FUNCTION_BLOCK Q_SelectColourMap (* Command Select Colour Map ( VT version 4 and later ) ( Part 6 - F.60 ) *)
  (* Standard: ISO 11783-6; Description: Copyright (c) 2022 HR Agrartechnik GmbH This program and the accompanying materials are made available under the terms of the Eclipse Public License 2.0 which is available at https://www.eclipse.org/legal/epl-2.0/ SPDX-License-Identifier: EPL-2.0 see Description Tab *)
  (* Version 1.0, 2022-07-08, Franz Höpfinger, HR Agrartechnik GmbH *)
  PACKAGE isobus::UT::Q;
  IMPORT isobus::UT::Q::const::IDs::ID_NULL;
  (* Documentation:
  Command Select Colour Map ( VT version 4 and later ) ( Part 6 - F.60 )
   The Select Colour Map command is used to select the active Colour Map. This command can take a long time to execute. The command applies to any presentation from the originating Working Set, which includes objects that may be shown on other Working Set screens (e.g. Auxiliary Control objects as may be presented on VT proprietary and other Working Set masks using the Auxiliary Control Designator Type 2 Object Pointer).
   Valid values for u16ObjIdColourMap
   The Select Colour Map or Palette command (F.60) carries, in bytes 2,3, the Object ID of the Colour Map object, the Colour Palette object, or FFFF16 to restore the default colour mapping (see A.3):
    - ColourMap: 39000 – 39999 (VT version 4 and later)
   - ColourPalette: 45000 – 45999 (VT version 6 and later, per Annex F.60)
   - FFFF16: restores the default colour table (see A.3)
    Implementation note (VTClientHelper): iso_is_colour_map_id only accepts the ColourMap range — a ColourPalette ID (45000 – 45999) is rejected. In addition, ID_NULL (65535), the documented FFFF16 value to restore the default colour table, is swallowed by cmd_select_colour_map_or_palette, which returns VT_E_NO_ERR (0) without sending any command to the VT. These are known deviations.
   param[in] {objectID, uint16_t}
   Object ID of Colour map object or FFFF to restore the default colour table (see A.3)
   Return Values (s16result):
   int16_t
    - VT_E_NO_ERR (0) - OK
   - VT_E_NOT_READY (-131) - VT client not yet ready
   - VT_E_OVERFLOW (-6) - buffer overflow
   - VT_E_NOACT (-8) - Command not possible in current state
   - VT_E_NO_INSTANCE (-21) - No VT client available
   - VT_E_ISO_INSTANCE_INVALID (-129) - Identifier for instance (connection) invalid
   - VT_E_NOT_ALIVE (-130) - Identifier for instance valid, but VT Dead.
   - VT_OK_BUFFERED (18) - command buffered, waiting for VT to be ready
    Instanz-Eindeutigkeit (Instance Uniqueness)
   Dieser Baustein ist konzeptionell als Singleton (genau eine Instanz im gesamten Programm) vorgesehen.
  *)
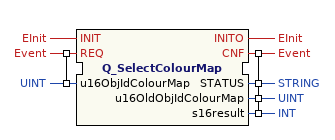
  EVENT_INPUT
    INIT : EInit; (* Service Initialization *)
    REQ WITH u16ObjIdColourMap; (* Service Request *)
  END_EVENT
  EVENT_OUTPUT
    INITO : EInit; (* Initialization Confirm *)
    CNF WITH STATUS, s16result, u16OldObjIdColourMap; (* Confirmation of Requested Service *)
  END_EVENT
  VAR_INPUT
    u16ObjIdColourMap : UINT := ID_NULL; (* Object ID of Colour map object or FFFF to restore the default colour table (see A.3) *)
  END_VAR
  VAR_OUTPUT
    STATUS : STRING; (* Service Status *)
    u16OldObjIdColourMap : UINT; (* Old object ID of Colour map object or FFFF to restore the default colour table (see A.3) *)
    s16result : INT; (* retval see description *)
  END_VAR
END_FUNCTION_BLOCK
